// Standard FS string.
// Size is a parameter located at FSParam_Core.nFST_STR_SIZE. | DEFAULT: 80
TYPE FsT_Str : STRING(FSParam_Core.STR_SIZE); END_TYPE

(* stored: Version 1.1.0.1, ProductVersion 3.1.4024.4
   DUT FsT_Str: Id {195d2a88-0bae-4800-a8d8-2e9f97a34e4f} *)
